FUNCTION_BLOCK StateMachine
VAR_INPUT	
END_VAR

VAR_OUTPUT
	bEntryConveyor		: BOOL := GVL.mb_Input_Coils[0];
	bBufferConveyor		: BOOL := GVL.mb_Input_Coils[1];
	bEmitter 			: BOOL := GVL.mb_Input_Coils[2];
END_VAR
VAR
	bItemReady			: BOOL := GVL.mb_Output_Coils[0];
	bAtEntry			: BOOL := GVL.mb_Output_Coils[1];
	bAtExit				: BOOL := GVL.mb_Output_Coils[2];	
	bFactoryIORunning 	: BOOL := GVL.mb_Output_Coils[3];
	bFactoryIOPaused 	: BOOL := GVL.mb_Output_Coils[4];
	bFactoryIOReset 	: BOOL := GVL.mb_Output_Coils[5];
END_VAR

// READ Inputs
	bItemReady			:= GVL.mb_Output_Coils[0];
	bAtEntry			:= GVL.mb_Output_Coils[1];
	bAtExit				:= GVL.mb_Output_Coils[2];	
	bFactoryIORunning 	:= GVL.mb_Output_Coils[3];
	bFactoryIOPaused 	:= GVL.mb_Output_Coils[4];
	bFactoryIOReset 	:= GVL.mb_Output_Coils[5];

// RESET	
IF bFactoryIOReset THEN
	GVL.iState := 0;
END_IF

// START Sequence
IF bFactoryIORunning AND NOT bFactoryIOPaused THEN
	CASE GVL.iState OF
		0:
			bEmitter:= TRUE;
			bEntryConveyor := TRUE;
			bBufferConveyor := FALSE;
			GVL.iState := 10; 
		10:
			
			bEntryConveyor := TRUE;
			IF NOT bItemReady THEN 	
				bEmitter := FALSE;		
				GVL.iState := 20;
			END_IF; 
		20:
			bEntryConveyor := TRUE;
			IF NOT bAtEntry THEN
				GVL.iState := 30;
			END_IF; 
		30:
			bEntryConveyor := TRUE;
			bBufferConveyor := TRUE;
			IF bAtEntry THEN
				GVL.iState := 40;
			END_IF; 
		40:
			bEntryConveyor := FALSE;
			bBufferConveyor := TRUE;
			IF NOT bAtExit THEN
				GVL.iState := 50;
			END_IF; 
		50:
			bEntryConveyor := FALSE;
			bBufferConveyor := TRUE;
			IF bAtExit THEN
				GVL.iState := 0;
			END_IF;
	END_CASE;
END_IF;

// WRITE OUTPUTS
	GVL.mb_Input_Coils[0]:= bEntryConveyor;
	GVL.mb_Input_Coils[1]:= bBufferConveyor;
	GVL.mb_Input_Coils[2]:= bEmitter;

END_FUNCTION_BLOCK

(* stored: Version 1.1.0.1, ProductVersion 3.1.4024.12
   POU StateMachine: Id {a7043d24-70f2-47a5-81ee-c765ce85ba4a}, SpecialFunc None *)
